// TIA Portal V20 export
TYPE "LER_typeUnitDataReelCut"
// stored: Access Published
   STRUCT
      Vision : "LER_typeVisionDataReelCut";
      QR_CutConveyor : "LER_typeQrData";
      QR_StackConveyor : "LER_typeQrData";
   END_STRUCT;
END_TYPE
